// TIA Portal V20 export
TYPE "typeCmControlNodeInterlock"
// stored: Namespace Unit1.Em3
   STRUCT
      masterVirtualAxis { ExternalWritable := 'False'} : "LER_typeAxisInterlock";
      unWinderVirtualAxis { ExternalWritable := 'False'} : "LER_typeAxisInterlock";
      dancerRegulator { ExternalWritable := 'False'} : "LER_typeTwoWayActuatorInterlock";
   END_STRUCT;
END_TYPE
